// TIA Portal V20 export
VAR_GLOBAL   // PLC tag table "Cabinet13"
   Sz13_Column_Red AT %Q1201.2 : Bool;
   Sz13_Column_Buzzer AT %Q1201.4 : Bool;
   Sz13_Column_Green AT %Q1200.6 : Bool;
   Sz13_Column_Yellow AT %Q1201.0 : Bool;
END_VAR
